FUNCTION_BLOCK ReactorSensors (* Composite Function Block Type *)
  (* Standard: 61499-2 *)
  (* Version 0.0, 11/14/2023, SESA371406, Schneider Electric, template *)
  PACKAGE SE.Nereda;
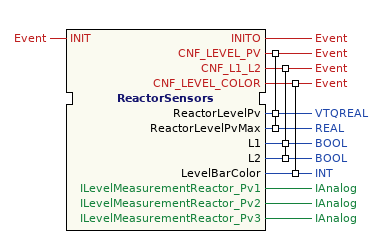
  EVENT_INPUT
    INIT; (* Initializes the symbolic link data destination FB with N (1 <= N <= 16) variables *)
  END_EVENT
  EVENT_OUTPUT
    INITO; (* Initialization Confirm *)
    CNF_LEVEL_PV WITH ReactorLevelPv, ReactorLevelPvMax; (* Execution confirmation of Pv *)
    CNF_L1_L2 WITH L1, L2;
    CNF_LEVEL_COLOR WITH LevelBarColor;
  END_EVENT
  VAR_OUTPUT
    ReactorLevelPv : VTQREAL; (* Scaled process signal *)
    ReactorLevelPvMax : REAL; (* Maximun pv measurement range (in engineering units) *)
    L1 : BOOL; (* Output event qualifier *)
    L2 : BOOL; (* Output event qualifier *)
    LevelBarColor : INT;
  END_VAR
  PLUGS
    ILevelMeasurementReactor_Pv1 : IAnalog; (* Process value and status interface adapter *)
    ILevelMeasurementReactor_Pv2 : IAnalog; (* Process value and status interface adapter *)
    ILevelMeasurementReactor_Pv3 : IAnalog; (* Process value and status interface adapter *)
  END_PLUGS
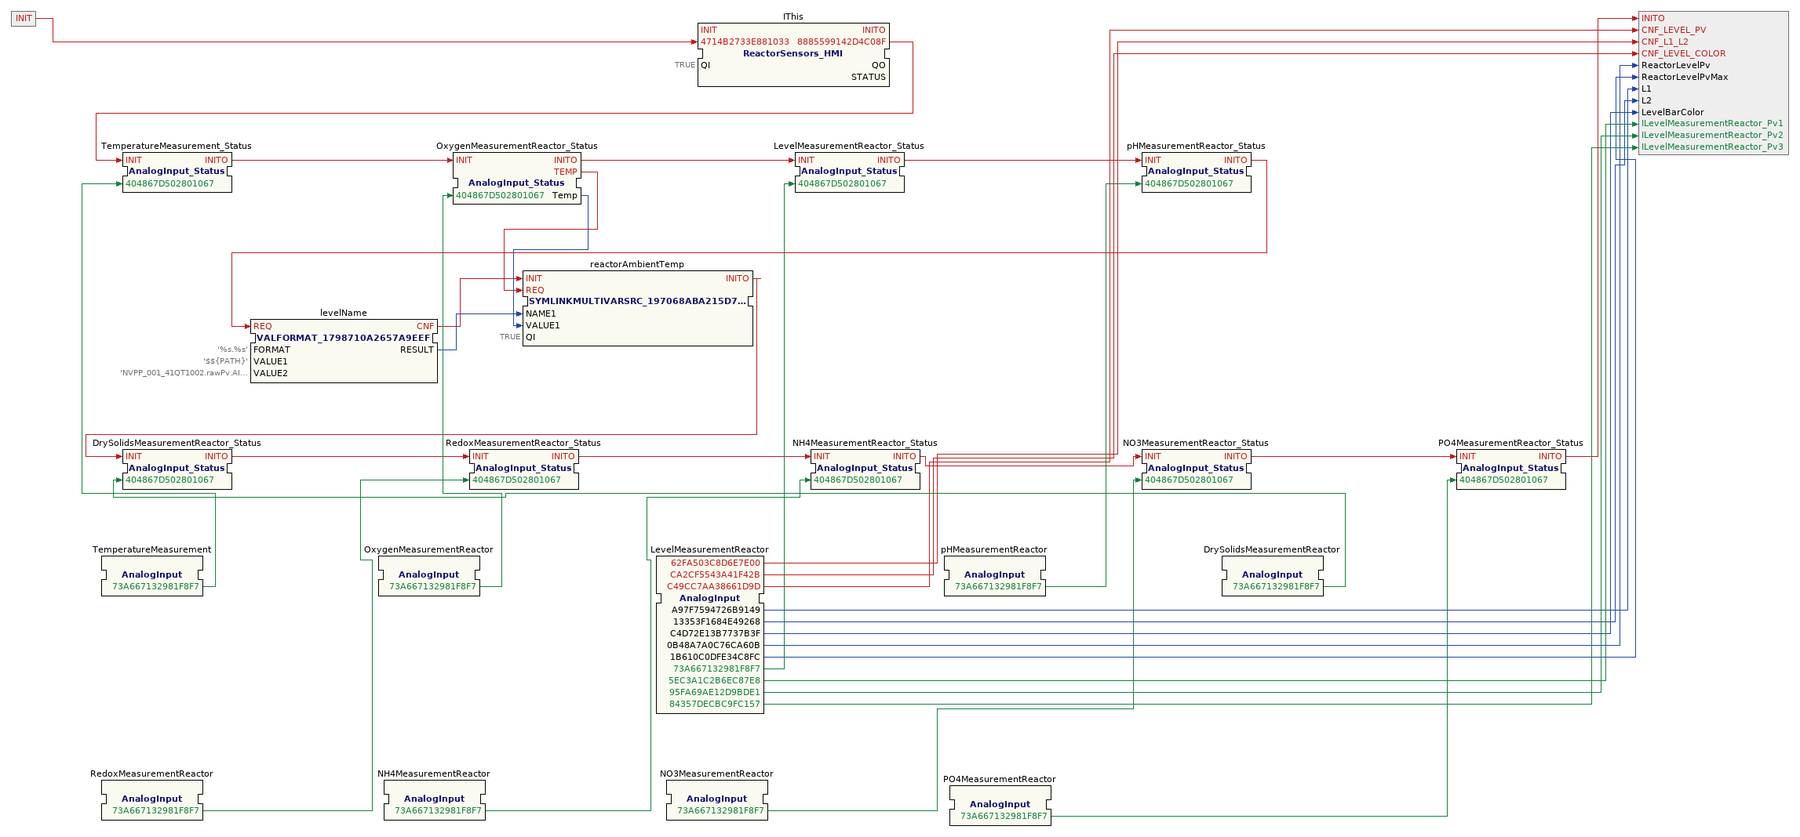
  (* 02 - FUNCTIONNAL OUTPUT INTERFACE *)
  (* HMI *)
  (* 01 - FUNCTIONNAL INPUT INTERFACE *)
  (* 00 - INITIALIZATION *)
  (* 05 - LOGIC *)
  (* 06 - HMI INTERFACE *)
  (* 02 - FUNCTIONNAL OUTPUT INTERFACE *)
  (* Actuators Status *)
  (* 03 - FIELD INTERFACE *)
  (* Temperature measurement *)
  (* Oxygen measurement reactor *)
  (* Level measurement reactor *)
  (* pH measurement reactor *)
  (* Dry solids measurement reactor *)
  (* Redox measurement reactor *)
  (* NH4 measurement reactor *)
  (* NO3 measurement reactor *)
  (* PO4 measurement reactor *)
  (* Add of the Valformat + SYMlink We had it as the reactor's Ambien temperature was shared through the SC1000_ AnalogInput so we are getting back the values and sharing it to the Ambinet temperature Analog Input by the symlink In the NVPP installation the reactor's ambient temperature sensor was not existing so we used that work aroud *)
  FBS
    TemperatureMeasurement_Status : AnalogInput_Status;
    pHMeasurementReactor_Status : AnalogInput_Status;
    OxygenMeasurementReactor_Status : AnalogInput_Status;
    LevelMeasurementReactor_Status : AnalogInput_Status;
    IThis : ReactorSensors_HMI(QI := TRUE);
    reactorAmbientTemp : SYMLINKMULTIVARSRC_197068ABA215D7EBA(QI := TRUE); {SET_ATTRIBUTE(Configuration.GenericFBType.InterfaceParams, Runtime.System#I:=1;VALUE${I$}:REAL)}
    levelName : VALFORMAT_1798710A2657A9EEF(FORMAT := '%s.%s', VALUE1 := '$${PATH}', VALUE2 := 'NVPP_001_41QT1002.rawPv.AIn'); {SET_ATTRIBUTE(Configuration.GenericFBType.InterfaceParams, Runtime.Standard#I:=2;VALUE${I$}:STRING,STRING)}
    TemperatureMeasurement : AnalogInput;
    OxygenMeasurementReactor : AnalogInput;
    LevelMeasurementReactor : AnalogInput;
    pHMeasurementReactor : AnalogInput;
    DrySolidsMeasurementReactor : AnalogInput;
    RedoxMeasurementReactor : AnalogInput;
    DrySolidsMeasurementReactor_Status : AnalogInput_Status;
    RedoxMeasurementReactor_Status : AnalogInput_Status;
    NH4MeasurementReactor : AnalogInput;
    NO3MeasurementReactor : AnalogInput;
    PO4MeasurementReactor : AnalogInput;
    NH4MeasurementReactor_Status : AnalogInput_Status;
    NO3MeasurementReactor_Status : AnalogInput_Status;
    PO4MeasurementReactor_Status : AnalogInput_Status;
  END_FBS
  EVENT_CONNECTIONS
    PO4MeasurementReactor_Status.INITO TO INITO;
    INIT TO IThis.4714B2733E881033;
    levelName.CNF TO reactorAmbientTemp.INIT;
    IThis.8885599142D4C08F TO TemperatureMeasurement_Status.INIT;
    TemperatureMeasurement_Status.INITO TO OxygenMeasurementReactor_Status.INIT;
    OxygenMeasurementReactor_Status.INITO TO LevelMeasurementReactor_Status.INIT;
    LevelMeasurementReactor_Status.INITO TO pHMeasurementReactor_Status.INIT;
    pHMeasurementReactor_Status.INITO TO levelName.REQ;
    LevelMeasurementReactor.62FA503C8D6E7E00 TO CNF_L1_L2;
    LevelMeasurementReactor.CA2CF5543A41F42B TO CNF_LEVEL_COLOR;
    LevelMeasurementReactor.C49CC7AA38661D9D TO CNF_LEVEL_PV;
    OxygenMeasurementReactor_Status.TEMP TO reactorAmbientTemp.REQ;
    DrySolidsMeasurementReactor_Status.INITO TO RedoxMeasurementReactor_Status.INIT;
    reactorAmbientTemp.INITO TO DrySolidsMeasurementReactor_Status.INIT;
    RedoxMeasurementReactor_Status.INITO TO NH4MeasurementReactor_Status.INIT;
    NH4MeasurementReactor_Status.INITO TO NO3MeasurementReactor_Status.INIT;
    NO3MeasurementReactor_Status.INITO TO PO4MeasurementReactor_Status.INIT;
  END_CONNECTIONS
  DATA_CONNECTIONS
    levelName.RESULT TO reactorAmbientTemp.NAME1;
    LevelMeasurementReactor.A97F7594726B9149 TO L1;
    LevelMeasurementReactor.13353F1684E49268 TO L2;
    LevelMeasurementReactor.C4D72E13B7737B3F TO LevelBarColor;
    LevelMeasurementReactor.0B48A7A0C76CA60B TO ReactorLevelPv;
    LevelMeasurementReactor.1B610C0DFE34C8FC TO ReactorLevelPvMax;
    OxygenMeasurementReactor_Status.Temp TO reactorAmbientTemp.VALUE1;
  END_CONNECTIONS
  ADAPTER_CONNECTIONS
    TemperatureMeasurement.73A667132981F8F7 TO TemperatureMeasurement_Status.404867D502801067;
    OxygenMeasurementReactor.73A667132981F8F7 TO OxygenMeasurementReactor_Status.404867D502801067;
    LevelMeasurementReactor.73A667132981F8F7 TO LevelMeasurementReactor_Status.404867D502801067;
    pHMeasurementReactor.73A667132981F8F7 TO pHMeasurementReactor_Status.404867D502801067;
    LevelMeasurementReactor.5EC3A1C2B6EC87E8 TO ILevelMeasurementReactor_Pv1;
    LevelMeasurementReactor.95FA69AE12D9BDE1 TO ILevelMeasurementReactor_Pv2;
    LevelMeasurementReactor.84357DECBC9FC157 TO ILevelMeasurementReactor_Pv3;
    DrySolidsMeasurementReactor.73A667132981F8F7 TO DrySolidsMeasurementReactor_Status.404867D502801067;
    RedoxMeasurementReactor.73A667132981F8F7 TO RedoxMeasurementReactor_Status.404867D502801067;
    NH4MeasurementReactor.73A667132981F8F7 TO NH4MeasurementReactor_Status.404867D502801067;
    NO3MeasurementReactor.73A667132981F8F7 TO NO3MeasurementReactor_Status.404867D502801067;
    PO4MeasurementReactor.73A667132981F8F7 TO PO4MeasurementReactor_Status.404867D502801067;
  END_CONNECTIONS
END_FUNCTION_BLOCK
